Staubli VAL3: ros_server.dtx

public bool bFbkOverrun
public bool bMotionOverrun
public sio siTcpIpFbk = {link=Serial\0}
public sio siTcpIpMotion = {link=Serial\0}
public string sStreamTaskName = "publisher"
public string sMotionTaskName
public RosSimpleMsg rosGenericMsg
  [0]
    Header header
      [0]
        num nMsgType
        num nCommType
        num nReplyCode
        num nData[12]
    Prefix prefix
      [0]
        num nLength
        num nData[4]
public tool tTool = {fatherId=flange[0], ioLink=valve1}
public string sTrajPtTaskName
public bool bTrajPtOverrun
public RobotStatusMsg rosStatusMsg
  [0]
    Body body
      [0]
        num nData[28]
    Header header
      [0]
        num nMsgType
        num nCommType
        num nReplyCode
        num nData[12]
    Prefix prefix
      [0]
        num nLength
        num nData[4]
    RobotStatus robotStatus
      [0]
        num nDrivesPowered
        num nEStopped
        num nErrorCode
        num nInError
        num nInMotion
        num nMode
        num nMotionPossible
public JointStateMsg rosJointMsg
  [0]
    Header header
      [0]
        num nMsgType
        num nCommType
        num nReplyCode
        num nData[12]
    Body body
      [0]
        num nData[44]
    JointState jointState
      [0]
        num nSeq
        num nJoints[10]
    Prefix prefix
      [0]
        num nLength
        num nData[4]
public JointTrajPtMsg rosTrajPtMsg
  [0]
    Header header
      [0]
        num nMsgType
        num nCommType
        num nReplyCode
        num nData[12]
    JointTrajPt jointTrajPt
      [0]
        num nSeq
        num nJoints[10]
        num nVelocity
        num nDuration
    Prefix prefix
      [0]
        num nLength
        num nData[4]
    Body body
      [0]
        num nData[52]
public JointTrajPtFMsg rosTrajPtFMsg
  [0]
    Header header
      [0]
        num nMsgType
        num nCommType
        num nReplyCode
        num nData[12]
    Prefix prefix
      [0]
        num nLength
        num nData[4]
    JointTrajPtFull jointTrajPtFull
      [0]
        num nRobotId
        num nSeq
        num nValidFields
        num nTime
        num nPositions[10]
        num nVelocities[10]
        num nAccelerations[10]
    Body body
      [0]
        num nData[136]
public JointFbkMsg rosJointFbkMsg
  [0]
    Header header
      [0]
        num nMsgType
        num nCommType
        num nReplyCode
        num nData[12]
    Prefix prefix
      [0]
        num nLength
        num nData[4]
    JointFeedback jointFeedback
      [0]
        num nRobotId
        num nValidFields
        num nTime
        num nPositions[10]
        num nVelocities[10]
        num nAccelerations[10]
    Body body
      [0]
        num nData[132]
public JointTrajPtFMsg rosTrajPtFAck
  [0]
    Header header
      [0]
        num nMsgType
        num nCommType
        num nReplyCode
        num nData[12]
    Prefix prefix
      [0]
        num nLength
        num nData[4]
    JointTrajPtFull jointTrajPtFull
      [0]
        num nRobotId
        num nSeq
        num nValidFields
        num nTime
        num nPositions[10]
        num nVelocities[10]
        num nAccelerations[10]
    Body body
      [0]
        num nData[136]
public JointTrajPtMsg rosTrajPtAck
  [0]
    Header header
      [0]
        num nMsgType
        num nCommType
        num nReplyCode
        num nData[12]
    JointTrajPt jointTrajPt
      [0]
        num nSeq
        num nJoints[10]
        num nVelocity
        num nDuration
    Prefix prefix
      [0]
        num nLength
        num nData[4]
    Body body
      [0]
        num nData[52]
public bool bScreenOverrun
public string sScreenTaskName
public num nInConnFlag
public num nOutConnFlag
public screen scDebug
public screen scMonitor
public string sHtbtTaskName
public num nPtsPopped
public bool bStopNow
public num nMotionProgress
public num nMoveId
public num nMovePts
public num nElapsedTime
public num nHeaderTime
public bool bOverwriteVel
public Queue qMoveBuffer
  [0]
    num nPush
    num nPop
    num nElems
    MotionCmd buffer[10]
      [0]
        mdesc mDesc = {leave=0, reach=0}
        num nDuration
        num nSequence
        jointRx jJointRx
      [1]
        mdesc mDesc = {leave=0, reach=0}
        num nDuration
        num nSequence
        jointRx jJointRx
      [2]
        mdesc mDesc = {leave=0, reach=0}
        num nDuration
        num nSequence
        jointRx jJointRx
      [3]
        mdesc mDesc = {leave=0, reach=0}
        num nDuration
        num nSequence
        jointRx jJointRx
      [4]
        mdesc mDesc = {leave=0, reach=0}
        num nDuration
        num nSequence
        jointRx jJointRx
      [5]
        mdesc mDesc = {leave=0, reach=0}
        num nDuration
        num nSequence
        jointRx jJointRx
      [6]
        mdesc mDesc = {leave=0, reach=0}
        num nDuration
        num nSequence
        jointRx jJointRx
      [7]
        mdesc mDesc = {leave=0, reach=0}
        num nDuration
        num nSequence
        jointRx jJointRx
      [8]
        mdesc mDesc = {leave=0, reach=0}
        num nDuration
        num nSequence
        jointRx jJointRx
      [9]
        mdesc mDesc = {leave=0, reach=0}
        num nDuration
        num nSequence
        jointRx jJointRx
public Queue qTrajPtBuffer
  [0]
    num nPush
    num nPop
    num nElems
    MotionCmd buffer[10]
      [0]
        mdesc mDesc = {leave=0, reach=0}
        num nDuration
        num nSequence
        jointRx jJointRx
      [1]
        mdesc mDesc = {leave=0, reach=0}
        num nDuration
        num nSequence
        jointRx jJointRx
      [2]
        mdesc mDesc = {leave=0, reach=0}
        num nDuration
        num nSequence
        jointRx jJointRx
      [3]
        mdesc mDesc = {leave=0, reach=0}
        num nDuration
        num nSequence
        jointRx jJointRx
      [4]
        mdesc mDesc = {leave=0, reach=0}
        num nDuration
        num nSequence
        jointRx jJointRx
      [5]
        mdesc mDesc = {leave=0, reach=0}
        num nDuration
        num nSequence
        jointRx jJointRx
      [6]
        mdesc mDesc = {leave=0, reach=0}
        num nDuration
        num nSequence
        jointRx jJointRx
      [7]
        mdesc mDesc = {leave=0, reach=0}
        num nDuration
        num nSequence
        jointRx jJointRx
      [8]
        mdesc mDesc = {leave=0, reach=0}
        num nDuration
        num nSequence
        jointRx jJointRx
      [9]
        mdesc mDesc = {leave=0, reach=0}
        num nDuration
        num nSequence
        jointRx jJointRx
num nVel[2]
num nGenericMsgType{}
  [JOINT_TRAJ_PT] = 11
  [JOINT_TRAJ_PT_FULL] = 14
  [SERVICE_REQUEST] = 2
mdesc mNomSpeed
num nMsgState{}
  [RecHeader] = {}
  [DecHeader] = 1
  [RecBody] = 2
  [DecBody] = 3
  [PushMotion] = 4
  [Ack] = 5
  [Reset] = {}
